(* Schneider Machine Expert - Basic project ProyekAkhir_Haritsyam Anshari_2106728414, file version 2.7.0.0 *)
(* ProjectInformations: Name=New project *)

HARDWARE
  Cpu 0: TM221CE16R
  EthernetConfiguration: NetworkName=M221, IpAllocationMode=FixedAddress, IpAddress=0.0.0.0, SubnetMask=0.0.0.0
  SerialLineConfiguration: Baud=Baud19200, Parity=ParityEven, DataBits=DataBits8, StopBits=StopBits1, PhysicalMedium=PhysicalMediumRs485, TransmissionMode=TransmissionModeModbusRtu, SlaveId=1, Addressing=SlaveAddressing
  MastTask: UsePeriodScanMode=false, PeriodScan=100
  FastTask: Period=255
  CpuBehavior: StartingMode=StartAsPreviousState, AutoSaveRamOnEeprom=true, WatchdogPeriod=250

SYMBOLS  (address, symbol, comment, settings)
  %M0         "FactoryIO Running"
  %M1         "Bases at entry 1"
  %M2         "Bases 1 - Busy"
  %M3         "Bases at exit 1 RS"
  %M4         "Bases at entry 2"
  %M5         "Bases 2 - Busy"
  %M6         "Bases at exit 2 RS"
  %M7         "Lids at entry 1"
  %M8         "Lids 1 - Busy"
  %M9         "Lids 1 at exit"
  %M10        "Lids at entry 2"
  %M11        "Lids 2 - Busy"
  %M12        "Lids 2 at exit"
  %M13        "Bases 1 Exit Diffuse"
  %M14        "Bases 2 Exit Diffuse"
  %M15        "Lids 1 Exit Diffuse"
  %M16        "Lids 2 Exit Diffuse"
  %M17        "Selector 1 - State 0"
  %M18        "Selector 1 - State 1"
  %M19        "Selector 2 - 0 State"
  %M20        "Selector 2 - 1 State"
  %M25        "Move Z"
  %M26        "Part Diffuse"
  %M27        "Bases Clamped"
  %M28        "Bases Diffuse (Assembler)"
  %M29        "Items Detected"
  %M30        "Lids Clamped"
  %M31        "Lids Diffuse As"
  %M32        "Bases 1 Raw Conveyor"
  %M33        "Bases 2 Raw Conveyor"
  %M34        "Bases Exit 1 Conv"
  %M35        "Bases Exit 2 Conv"
  %M36        "Bases 1 Start"
  %M38        "Bases 1 Stop"
  %M39        "Bases 2 Start"
  %M41        "Bases 2 Stop"
  %M44        "Lids 1 Produce Lids"
  %M45        "Lids 2 Produce Lids"
  %M46        "Lids 1 Raw Conv"
  %M47        "Lids 2 Raw Conv"
  %M48        "Lids 1 - Start"
  %M49        "Lids 1 Reset"
  %M50        "Lids 1 Stop"
  %M51        "Lids 2 - Start"
  %M52        "Lids 2 Reset"
  %M53        "Lids 2 Stop"
  %M54        "Lids 1 Exit Conv"
  %M55        "Lids 2 Exit Conv"
  %M56        "Bases Belt Main 1"
  %M57        "Bases Belt Main 2"
  %M58        "Bases Belt Main 3"
  %M59        "Lids Belt Main 1"
  %M60        "Lids Belt Main 2"
  %M61        "Lids Belt Main 3"
  %M62        "Bases Blue Indicator"
  %M63        "Bases Green Indicator"
  %M64        "Lids Blue Indicator"
  %M65        "Lids Green Indicator"
  %M66        "Bases Assembler Conv"
  %M67        "Lids Assembler Conv"
  %M68        "Move Z"
  %M69        "Move X"
  %M70        "Grab"
  %M71        "Bases Clamp"
  %M72        "Lids Clamp"
  %M73        "Raise"
  %M74        "Base emitter 1"
  %M75        "Base emitter 2"
  %M76        "Lids emitter 1"
  %M77        "Lids emitter 2"
  %M78        "Remover"
  %TM0        [Type=TP, Preset=3, Base=OneSecond]
  %TM1        [Type=TP, Preset=1, Base=OneSecond]
  %TM2        [Preset=1, Base=OneSecond]
  %TM3        [Preset=1, Base=OneSecond]
  %TM4        [Type=TP, Preset=1, Base=OneSecond]
  %TM5        [Type=TP, Preset=3, Base=OneSecond]
  %TM6        [Preset=3, Base=OneSecond]
  %TM7        [Type=TP, Preset=2, Base=OneSecond]
  %TM8        [Type=TP, Preset=45, Base=OneHundredMilliSeconds]
  %TM9        [Type=TP, Preset=45, Base=OneHundredMilliSeconds]
  %TM10       [Type=TP, Preset=45, Base=OneHundredMilliSeconds]
  %TM11       [Type=TP, Preset=45, Base=OneHundredMilliSeconds]
  %Q0.0       "0_Memory_Bases"
  %Q0.1       "1_Memory_Lids"

POU New POU
  (* SectionNumber=1 *)

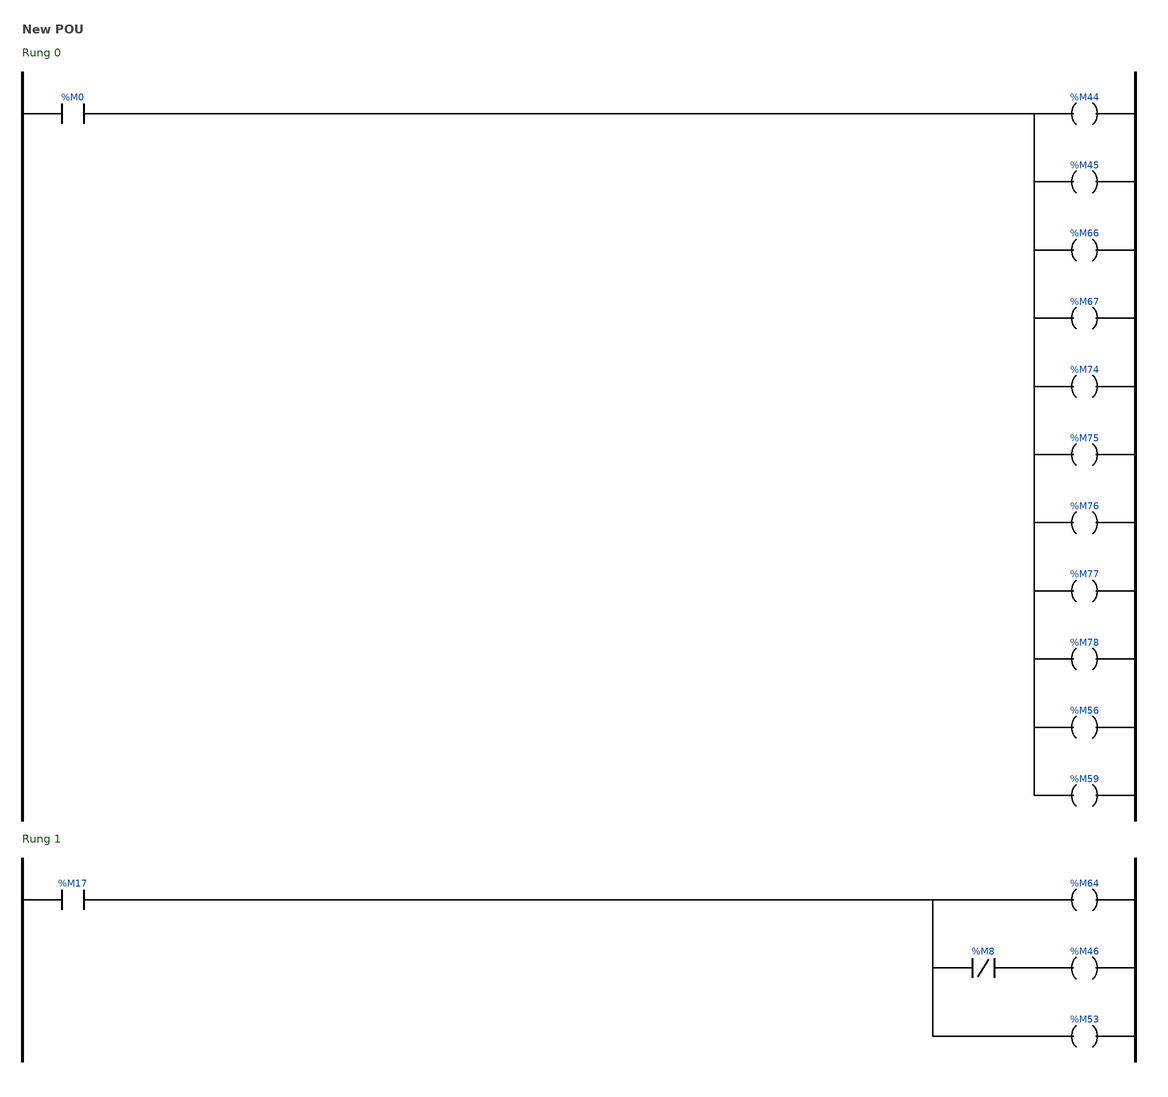

// Rung 0
  LD %M0
  ST %M44
  ST %M45
  ST %M66
  ST %M67
  ST %M74
  ST %M75
  ST %M76
  ST %M77
  ST %M78
  ST %M56
  ST %M59
  // as ST:
  //   %M44 := %M0;
  //   %M45 := %M0;
  //   %M66 := %M0;
  //   %M67 := %M0;
  //   %M74 := %M0;
  //   %M75 := %M0;
  //   %M76 := %M0;
  //   %M77 := %M0;
  //   %M78 := %M0;
  //   %M56 := %M0;
  //   %M59 := %M0;

// Rung 1
  LD %M17
  MPS
  ST %M64
  MRD
  ANDN %M8
  ST %M46
  MPP
  ST %M53
  // as ST:
  //   %M64 := %M17;
  //   %M46 := %M17 AND NOT %M8;
  //   %M53 := %M17;

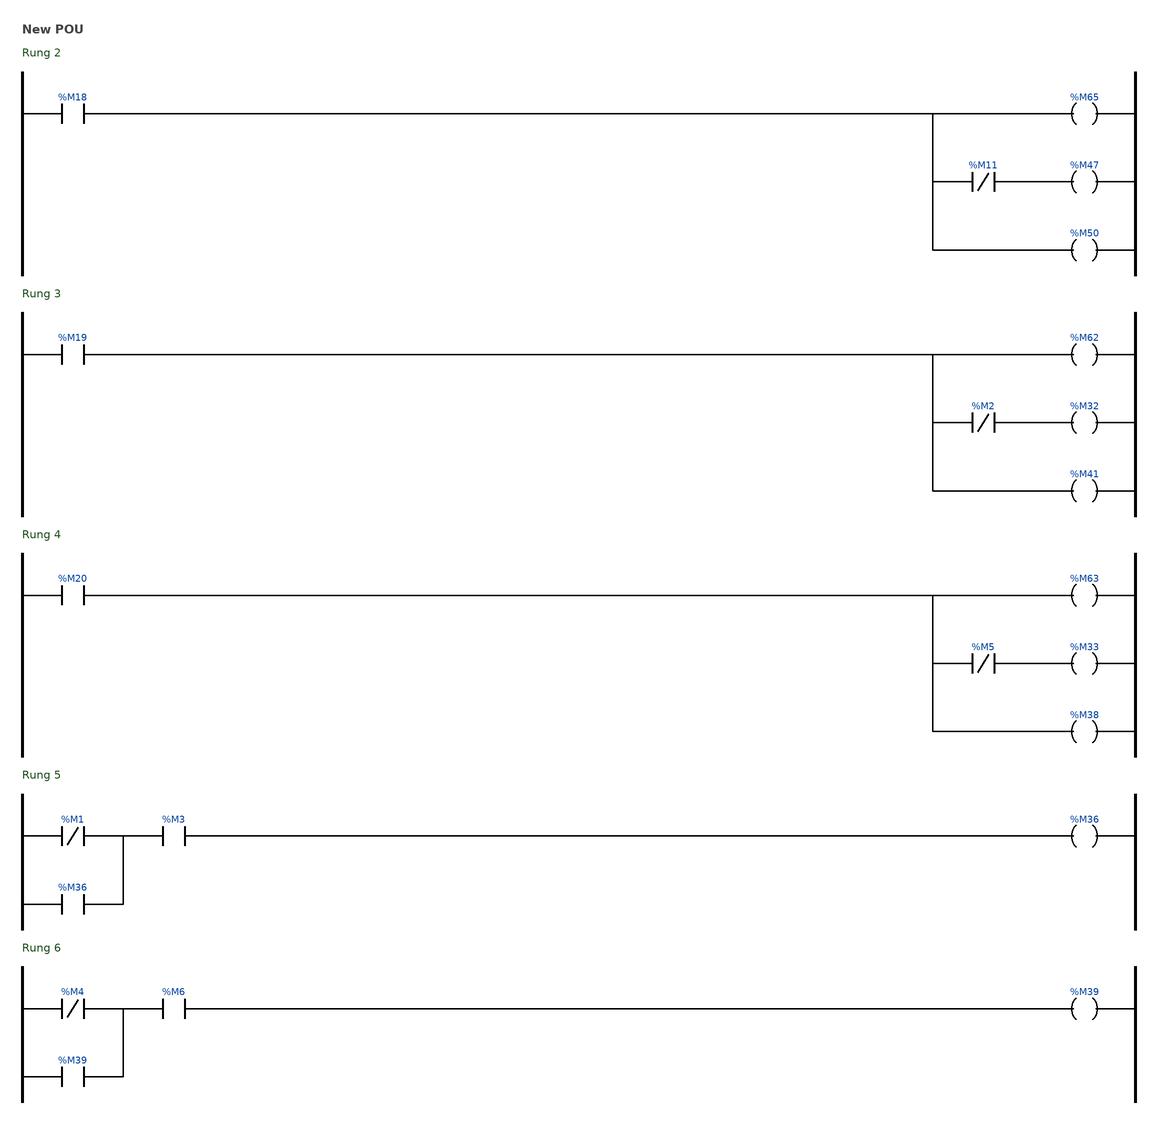

// Rung 2
  LD %M18
  MPS
  ST %M65
  MRD
  ANDN %M11
  ST %M47
  MPP
  ST %M50
  // as ST:
  //   %M65 := %M18;
  //   %M47 := %M18 AND NOT %M11;
  //   %M50 := %M18;

// Rung 3
  LD %M19
  MPS
  ST %M62
  MRD
  ANDN %M2
  ST %M32
  MPP
  ST %M41
  // as ST:
  //   %M62 := %M19;
  //   %M32 := %M19 AND NOT %M2;
  //   %M41 := %M19;

// Rung 4
  LD %M20
  MPS
  ST %M63
  MRD
  ANDN %M5
  ST %M33
  MPP
  ST %M38
  // as ST:
  //   %M63 := %M20;
  //   %M33 := %M20 AND NOT %M5;
  //   %M38 := %M20;

// Rung 5
  LDN %M1
  OR %M36
  AND %M3
  ST %M36
  // as ST:
  //   %M36 := (NOT %M1 OR %M36) AND %M3;

// Rung 6
  LDN %M4
  OR %M39
  AND %M6
  ST %M39
  // as ST:
  //   %M39 := (NOT %M4 OR %M39) AND %M6;

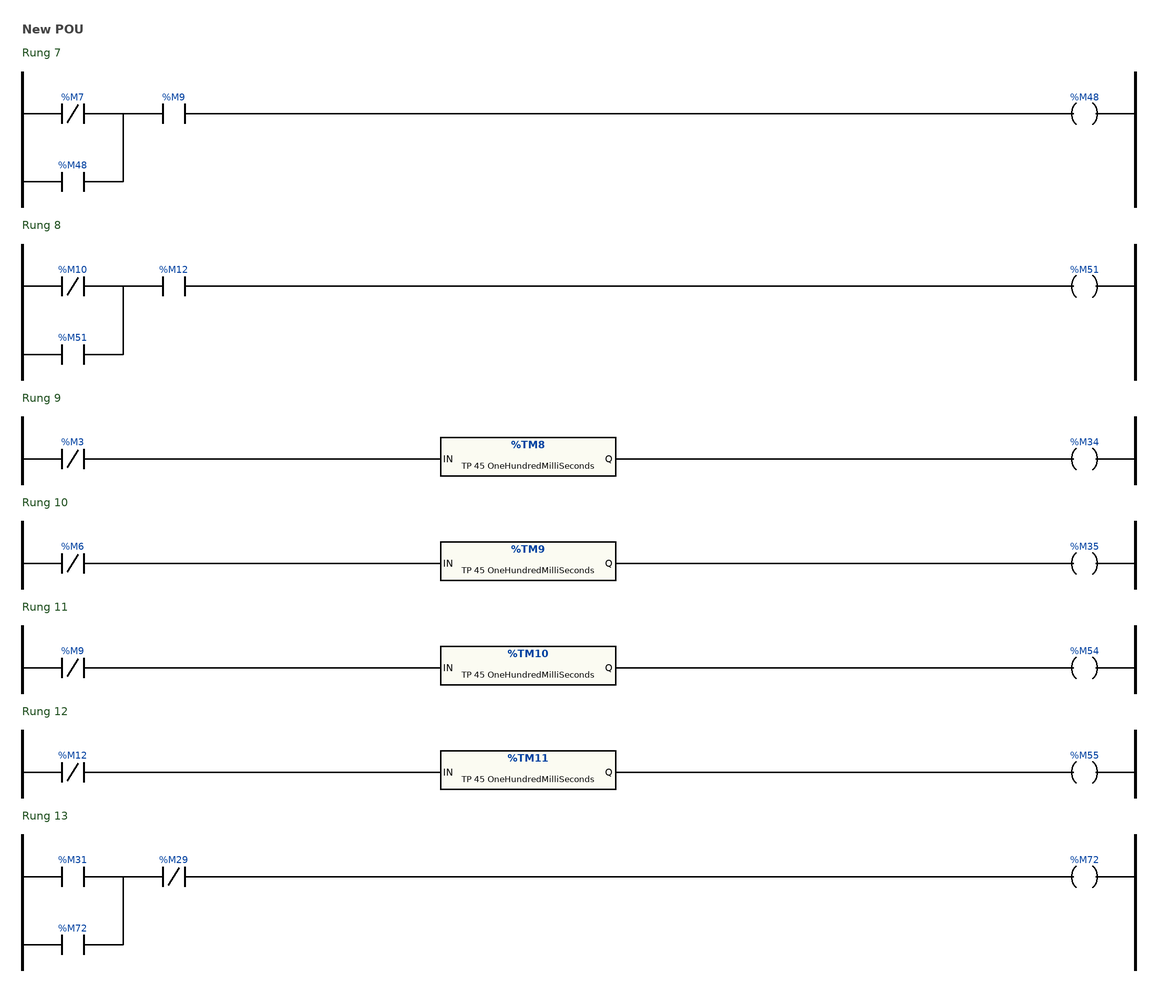

// Rung 7
  LDN %M7
  OR %M48
  AND %M9
  ST %M48
  // as ST:
  //   %M48 := (NOT %M7 OR %M48) AND %M9;

// Rung 8
  LDN %M10
  OR %M51
  AND %M12
  ST %M51
  // as ST:
  //   %M51 := (NOT %M10 OR %M51) AND %M12;

// Rung 9
  BLK %TM8
  LDN %M3
  IN
  OUT_BLK
  LD Q
  ST %M34
  END_BLK
  // as ST:
  //   %TM8(IN := NOT %M3);
  //   %M34 := %TM8.Q;

// Rung 10
  BLK %TM9
  LDN %M6
  IN
  OUT_BLK
  LD Q
  ST %M35
  END_BLK
  // as ST:
  //   %TM9(IN := NOT %M6);
  //   %M35 := %TM9.Q;

// Rung 11
  BLK %TM10
  LDN %M9
  IN
  OUT_BLK
  LD Q
  ST %M54
  END_BLK
  // as ST:
  //   %TM10(IN := NOT %M9);
  //   %M54 := %TM10.Q;

// Rung 12
  BLK %TM11
  LDN %M12
  IN
  OUT_BLK
  LD Q
  ST %M55
  END_BLK
  // as ST:
  //   %TM11(IN := NOT %M12);
  //   %M55 := %TM11.Q;

// Rung 13
  LD %M31
  OR %M72
  ANDN %M29
  ST %M72
  // as ST:
  //   %M72 := (%M31 OR %M72) AND NOT %M29;

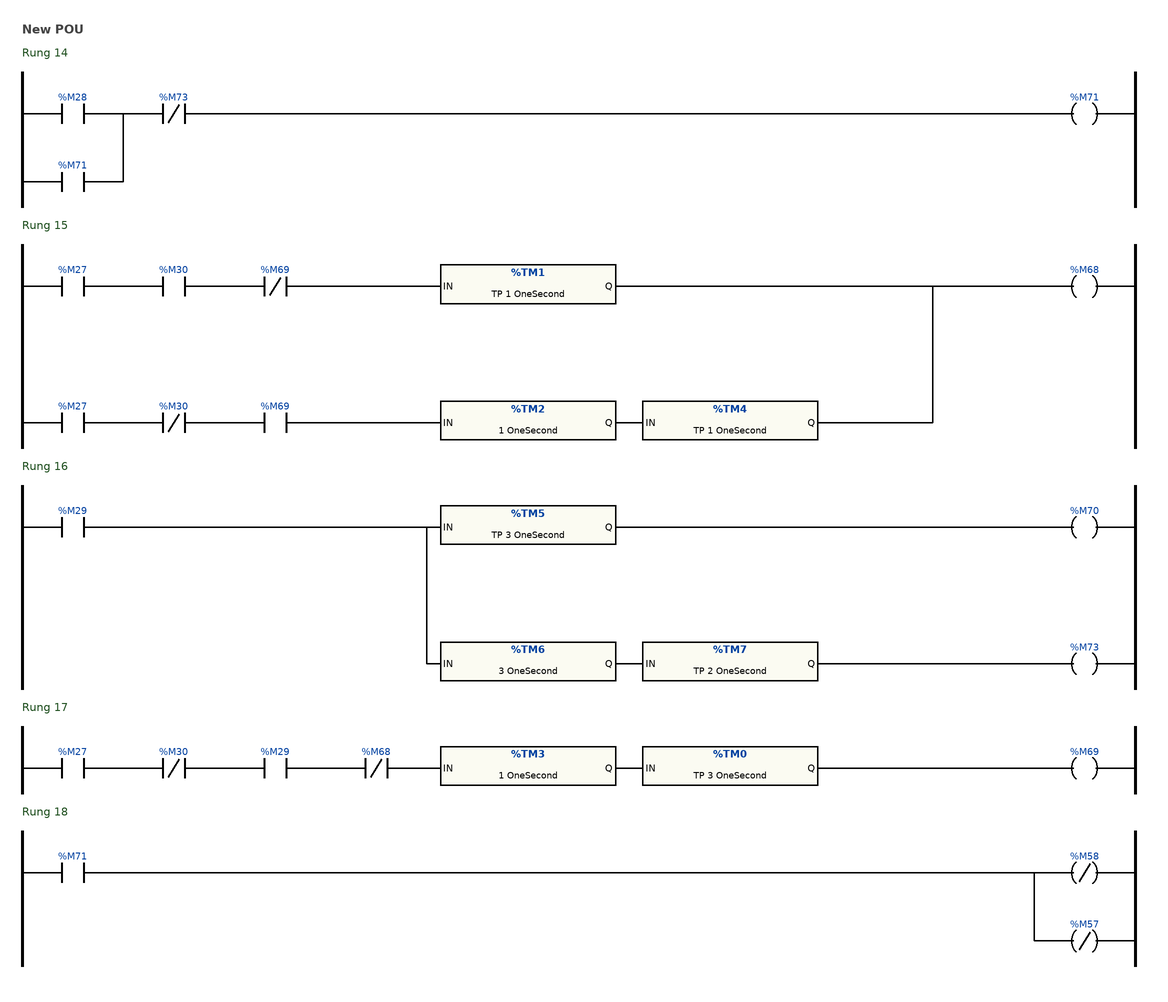

// Rung 14
  LD %M28
  OR %M71
  ANDN %M73
  ST %M71
  // as ST:
  //   %M71 := (%M28 OR %M71) AND NOT %M73;

// Rung 15
  LD 1
  MULTIFB
  LD 1
  ST %MW2009:X3
  BLK %TM1
  LD %MW2009:X3
  AND %M27
  AND %M30
  ANDN %M69
  IN
  OUT_BLK
  LD Q
  ST %MW2009:X0
  END_BLK
  BLK %TM2
  LD %MW2009:X3
  AND %M27
  ANDN %M30
  AND %M69
  IN
  OUT_BLK
  LD Q
  ST %MW2009:X1
  END_BLK
  BLK %TM4
  LD %MW2009:X1
  IN
  OUT_BLK
  LD Q
  ST %MW2009:X2
  END_BLK
  LD %MW2009:X0
  OR %MW2009:X2
  ST %M68
  MULTIFB
  // as ST:
  //   %TM1(IN := %M27 AND %M30 AND NOT %M69);
  //   %TM2(IN := %M27 AND NOT %M30 AND %M69);
  //   %TM4(IN := %TM2.Q);
  //   %M68 := %TM1.Q OR %TM4.Q;

// Rung 16
  LD 1
  MULTIFB
  LD 1
  AND %M29
  ST %MW2009:X1
  BLK %TM5
  LD %MW2009:X1
  IN
  OUT_BLK
  LD Q
  ST %M70
  END_BLK
  BLK %TM6
  LD %MW2009:X1
  IN
  OUT_BLK
  LD Q
  ST %MW2009:X0
  END_BLK
  BLK %TM7
  LD %MW2009:X0
  IN
  OUT_BLK
  LD Q
  ST %M73
  END_BLK
  MULTIFB
  // as ST:
  //   %TM5(IN := %M29);
  //   %M70 := %TM5.Q;
  //   %TM6(IN := %M29);
  //   %TM7(IN := %TM6.Q);
  //   %M73 := %TM7.Q;

// Rung 17
  LD 1
  MULTIFB
  BLK %TM3
  LD 1
  AND %M27
  ANDN %M30
  AND %M29
  ANDN %M68
  IN
  OUT_BLK
  LD Q
  ST %MW2009:X0
  END_BLK
  BLK %TM0
  LD %MW2009:X0
  IN
  OUT_BLK
  LD Q
  ST %M69
  END_BLK
  MULTIFB
  // as ST:
  //   %TM3(IN := %M27 AND NOT %M30 AND %M29 AND NOT %M68);
  //   %TM0(IN := %TM3.Q);
  //   %M69 := %TM0.Q;

// Rung 18
  LD %M71
  STN %M58
  STN %M57
  // as ST:
  //   %M58 := NOT %M71;
  //   %M57 := NOT %M71;

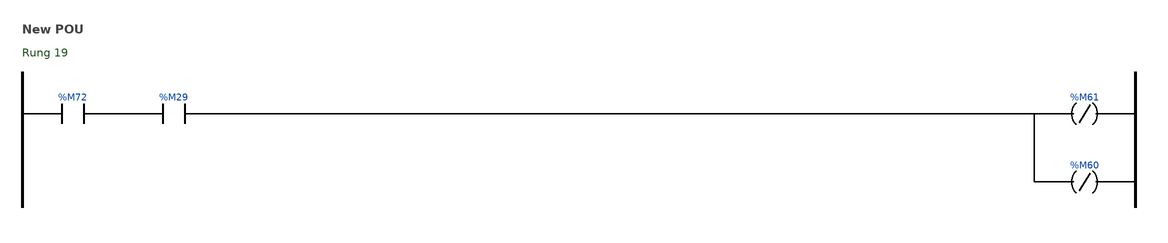

// Rung 19
  LD %M72
  AND %M29
  STN %M61
  STN %M60
  // as ST:
  //   %M61 := NOT (%M72 AND %M29);
  //   %M60 := NOT (%M72 AND %M29);
